Omron CX-Programmer project NewProject (CX-Programmer 9.75)

# PLC NewPLC1: CP1L M

## Global symbols (name address type ; comment)
0.00 BOOL  ; Penjumlahan
0.01 BOOL  ; Pengurangan
0.02 BOOL  ; Perkalian
0.03 BOOL  ; Pembagian

## Program NewProgram1 (cyclic task 0)

### Section Section1

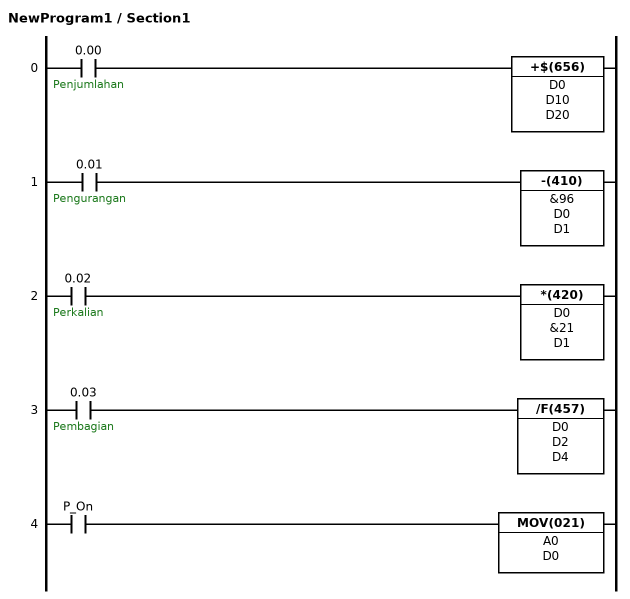
; rung 0
LD 0.00  ; Penjumlahan
+$(656) D0 D10 D20
; rung 1
LD 0.01  ; Pengurangan
-(410) &96 D0 D1
; rung 2
LD 0.02  ; Perkalian
*(420) D0 &21 D1
; rung 3
LD 0.03  ; Pembagian
/F(457) D0 D2 D4
; rung 4
LD P_On
MOV(021) A0 D0

### Section END
; rung 0
END(001)